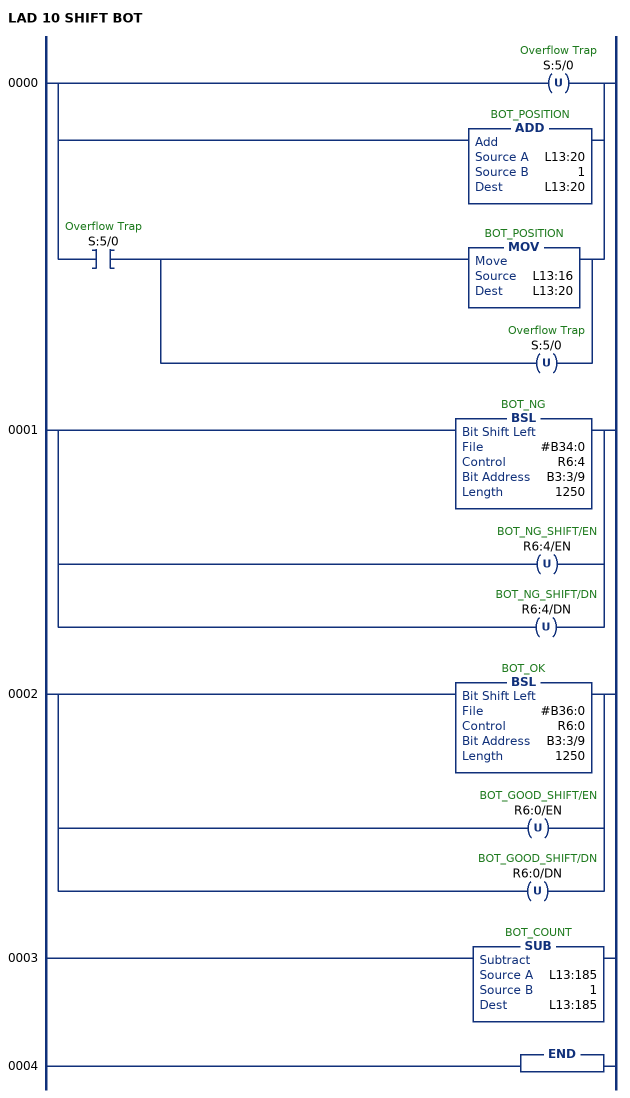
% Rung: 0 %
SOR BST OTU S:5/0 NXB ADD L13:20 1 L13:20 NXB XIC S:5/0 BST MOV L13:16 L13:20 NXB OTU S:5/0 BND BND EOR
%   S:5/0  "Overflow Trap" %
%   L13:20  BOT_POSITION %
%   L13:16  MIN_LONG %
% Rung: 1 %
SOR BST BSL #B34:0 R6:4 B3:3/9 1250 NXB OTU R6:4/EN NXB OTU R6:4/DN BND EOR
%   B34:0  BOT_NG %
%   R6:4  BOT_NG_SHIFT %
%   B3:3/9  OFF %
% Rung: 2 %
SOR BST BSL #B36:0 R6:0 B3:3/9 1250 NXB OTU R6:0/EN NXB OTU R6:0/DN BND EOR
%   B36:0  BOT_OK %
%   R6:0  BOT_GOOD_SHIFT %
%   B3:3/9  OFF %
% Rung: 3 %
SOR SUB L13:185 1 L13:185 EOR
%   L13:185  BOT_COUNT %
% Rung: 4 %
SOR END EOR

LADDER 11 "SHIFT TOP"
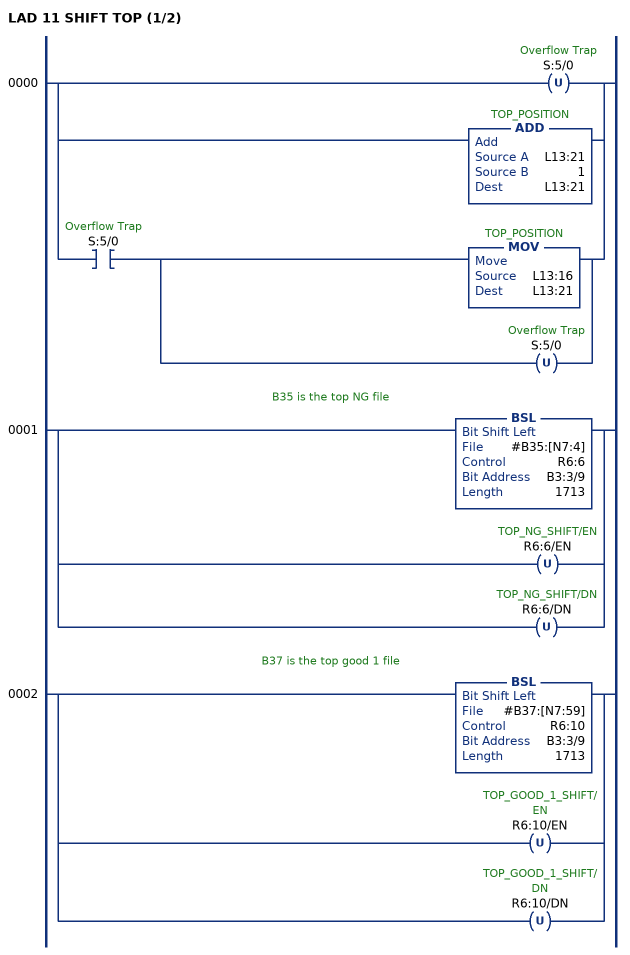
% Rung: 0 %
SOR BST OTU S:5/0 NXB ADD L13:21 1 L13:21 NXB XIC S:5/0 BST MOV L13:16 L13:21 NXB OTU S:5/0 BND BND EOR
%   S:5/0  "Overflow Trap" %
%   L13:21  TOP_POSITION %
%   L13:16  MIN_LONG %
% Rung: 1 %
% B35 is the top NG file %
SOR BST BSL #B35:[N7:4] R6:6 B3:3/9 1713 NXB OTU R6:6/EN NXB OTU R6:6/DN BND EOR
%   N7:4  TOP_NG_START_WORD %
%   R6:6  TOP_NG_SHIFT %
%   B3:3/9  OFF %
% Rung: 2 %
% B37 is the top good 1 file %
SOR BST BSL #B37:[N7:59] R6:10 B3:3/9 1713 NXB OTU R6:10/EN NXB OTU R6:10/DN BND EOR
%   N7:59  TOP_GOOD1_START_WORD %
%   R6:10  TOP_GOOD_1_SHIFT %
%   B3:3/9  OFF %

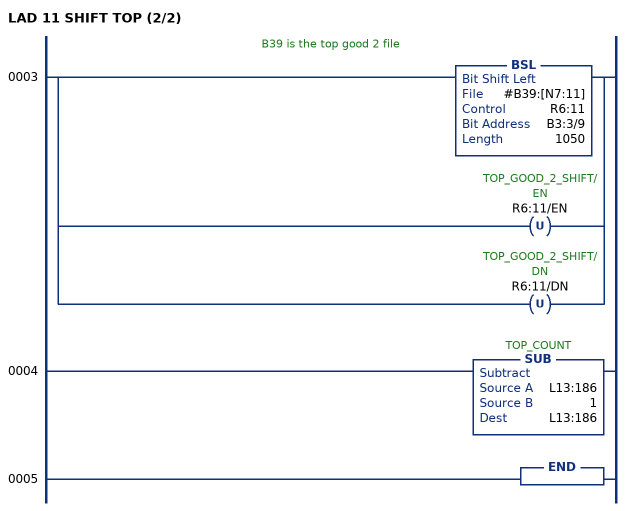
% Rung: 3 %
% B39 is the top good 2 file %
SOR BST BSL #B39:[N7:11] R6:11 B3:3/9 1050 NXB OTU R6:11/EN NXB OTU R6:11/DN BND EOR
%   N7:11  TOP_GOOD2_START_WORD %
%   R6:11  TOP_GOOD_2_SHIFT %
%   B3:3/9  OFF %
% Rung: 4 %
SOR SUB L13:186 1 L13:186 EOR
%   L13:186  TOP_COUNT %
% Rung: 5 %
SOR END EOR

LADDER 12 "BOTOPTIC"
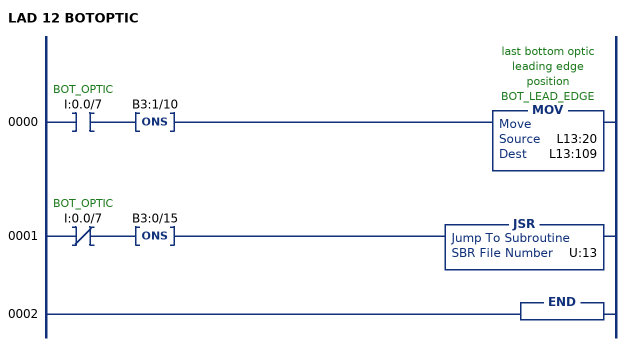
% Rung: 0 %
SOR XIC I:0.0/7 ONS B3:1/10 MOV L13:20 L13:109 EOR
%   I:0.0/7  BOT_OPTIC %
%   L13:20  BOT_POSITION %
%   L13:109  BOT_LEAD_EDGE  "last bottom optic leading edge position" %
% Rung: 1 %
SOR XIO I:0.0/7 ONS B3:0/15 JSR U:13 EOR
%   I:0.0/7  BOT_OPTIC %
% Rung: 2 %
SOR END EOR

LADDER 13 "BOTOPTMES"
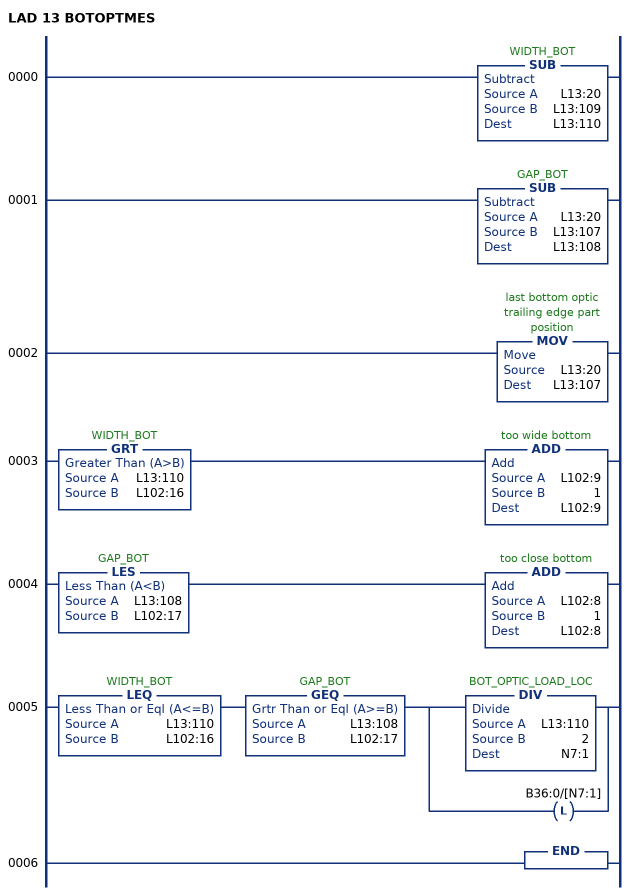
% Rung: 0 %
SOR SUB L13:20 L13:109 L13:110 EOR
%   L13:20  BOT_POSITION %
%   L13:109  BOT_LEAD_EDGE  "last bottom optic leading edge position" %
%   L13:110  WIDTH_BOT %
% Rung: 1 %
SOR SUB L13:20 L13:107 L13:108 EOR
%   L13:20  BOT_POSITION %
%   L13:107  "last bottom optic trailing edge part position" %
%   L13:108  GAP_BOT %
% Rung: 2 %
SOR MOV L13:20 L13:107 EOR
%   L13:20  BOT_POSITION %
%   L13:107  "last bottom optic trailing edge part position" %
% Rung: 3 %
SOR GRT L13:110 L102:16 ADD L102:9 1 L102:9 EOR
%   L13:110  WIDTH_BOT %
%   L102:16  BOT_MAX_WIDTH %
%   L102:9  "too wide bottom" %
% Rung: 4 %
SOR LES L13:108 L102:17 ADD L102:8 1 L102:8 EOR
%   L13:108  GAP_BOT %
%   L102:17  BOT_MIN_GAP %
%   L102:8  "too close bottom" %
% Rung: 5 %
SOR LEQ L13:110 L102:16 GEQ L13:108 L102:17 BST DIV L13:110 2 N7:1 NXB OTL B36:0/[N7:1] BND EOR
%   L13:110  WIDTH_BOT %
%   L102:16  BOT_MAX_WIDTH %
%   L13:108  GAP_BOT %
%   L102:17  BOT_MIN_GAP %
%   N7:1  BOT_OPTIC_LOAD_LOC %
%   B36:0  BOT_OK %
% Rung: 6 %
SOR END EOR

LADDER 14 "SHIFT TOP2"    % shift top inspection 6 %
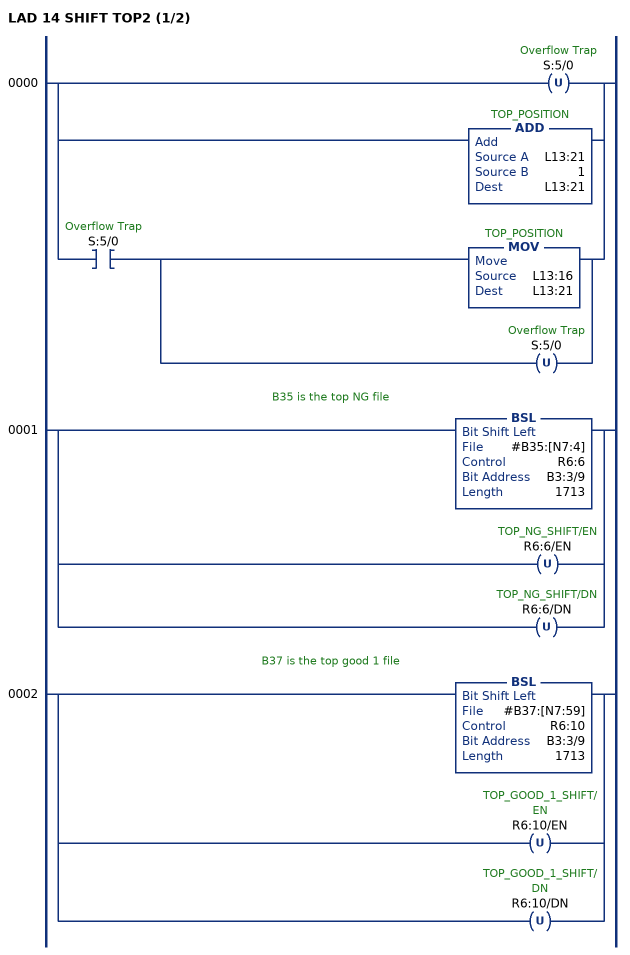
% Rung: 0 %
SOR BST OTU S:5/0 NXB ADD L13:21 1 L13:21 NXB XIC S:5/0 BST MOV L13:16 L13:21 NXB OTU S:5/0 BND BND EOR
%   S:5/0  "Overflow Trap" %
%   L13:21  TOP_POSITION %
%   L13:16  MIN_LONG %
% Rung: 1 %
% B35 is the top NG file %
SOR BST BSL #B35:[N7:4] R6:6 B3:3/9 1713 NXB OTU R6:6/EN NXB OTU R6:6/DN BND EOR
%   N7:4  TOP_NG_START_WORD %
%   R6:6  TOP_NG_SHIFT %
%   B3:3/9  OFF %
% Rung: 2 %
% B37 is the top good 1 file %
SOR BST BSL #B37:[N7:59] R6:10 B3:3/9 1713 NXB OTU R6:10/EN NXB OTU R6:10/DN BND EOR
%   N7:59  TOP_GOOD1_START_WORD %
%   R6:10  TOP_GOOD_1_SHIFT %
%   B3:3/9  OFF %

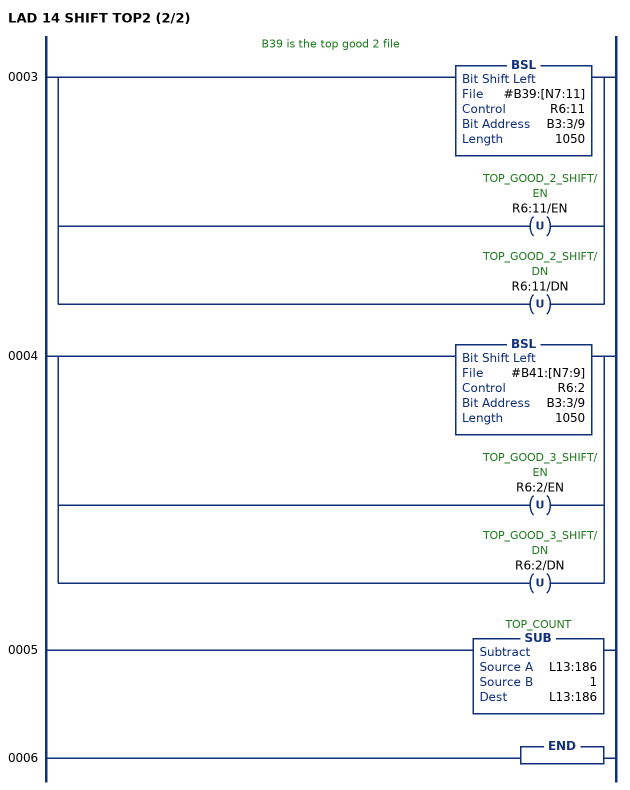
% Rung: 3 %
% B39 is the top good 2 file %
SOR BST BSL #B39:[N7:11] R6:11 B3:3/9 1050 NXB OTU R6:11/EN NXB OTU R6:11/DN BND EOR
%   N7:11  TOP_GOOD2_START_WORD %
%   R6:11  TOP_GOOD_2_SHIFT %
%   B3:3/9  OFF %
% Rung: 4 %
SOR BST BSL #B41:[N7:9] R6:2 B3:3/9 1050 NXB OTU R6:2/EN NXB OTU R6:2/DN BND EOR
%   N7:9  TOP_GOOD3_START_WORD %
%   R6:2  TOP_GOOD_3_SHIFT %
%   B3:3/9  OFF %
% Rung: 5 %
SOR SUB L13:186 1 L13:186 EOR
%   L13:186  TOP_COUNT %
% Rung: 6 %
SOR END EOR

LADDER 81 "I1"
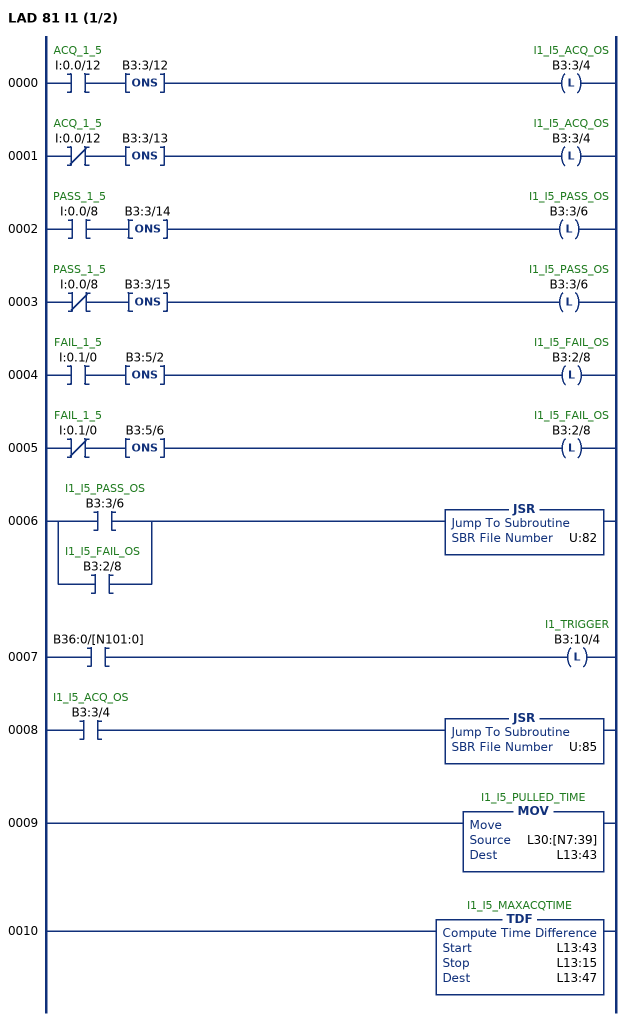
% Rung: 0 %
SOR XIC I:0.0/12 ONS B3:3/12 OTL B3:3/4 EOR
%   I:0.0/12  ACQ_1_5 %
%   B3:3/4  I1_I5_ACQ_OS %
% Rung: 1 %
SOR XIO I:0.0/12 ONS B3:3/13 OTL B3:3/4 EOR
%   I:0.0/12  ACQ_1_5 %
%   B3:3/4  I1_I5_ACQ_OS %
% Rung: 2 %
SOR XIC I:0.0/8 ONS B3:3/14 OTL B3:3/6 EOR
%   I:0.0/8  PASS_1_5 %
%   B3:3/6  I1_I5_PASS_OS %
% Rung: 3 %
SOR XIO I:0.0/8 ONS B3:3/15 OTL B3:3/6 EOR
%   I:0.0/8  PASS_1_5 %
%   B3:3/6  I1_I5_PASS_OS %
% Rung: 4 %
SOR XIC I:0.1/0 ONS B3:5/2 OTL B3:2/8 EOR
%   I:0.1/0  FAIL_1_5 %
%   B3:2/8  I1_I5_FAIL_OS %
% Rung: 5 %
SOR XIO I:0.1/0 ONS B3:5/6 OTL B3:2/8 EOR
%   I:0.1/0  FAIL_1_5 %
%   B3:2/8  I1_I5_FAIL_OS %
% Rung: 6 %
SOR BST XIC B3:3/6 NXB XIC B3:2/8 BND JSR U:82 EOR
%   B3:3/6  I1_I5_PASS_OS %
%   B3:2/8  I1_I5_FAIL_OS %
% Rung: 7 %
SOR XIC B36:0/[N101:0] OTL B3:10/4 EOR
%   B36:0  BOT_OK %
%   N101:0  I1_TRIG_LOC %
%   B3:10/4  I1_TRIGGER %
% Rung: 8 %
SOR XIC B3:3/4 JSR U:85 EOR
%   B3:3/4  I1_I5_ACQ_OS %
% Rung: 9 %
SOR MOV L30:[N7:39] L13:43 EOR
%   N7:39  I5_OLDEST_PART_INDEX %
%   L13:43  I1_I5_PULLED_TIME %
% Rung: 10 %
SOR TDF L13:43 L13:15 L13:47 EOR
%   L13:43  I1_I5_PULLED_TIME %
%   L13:15  THE_TIME %
%   L13:47  I1_I5_MAXACQTIME %

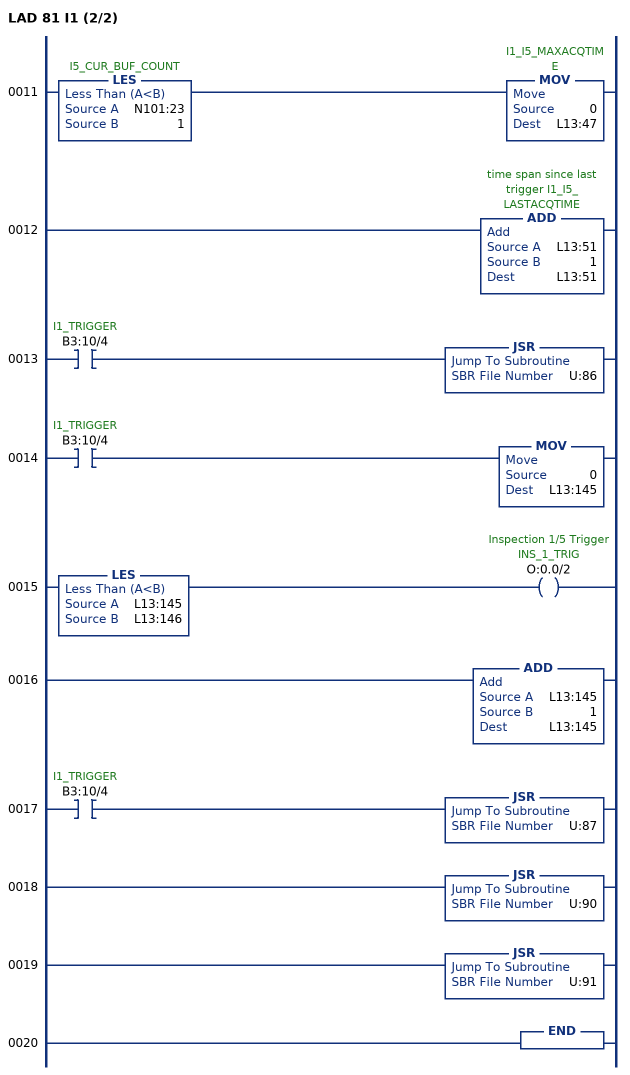
% Rung: 11 %
SOR LES N101:23 1 MOV 0 L13:47 EOR
%   N101:23  I5_CUR_BUF_COUNT %
%   L13:47  I1_I5_MAXACQTIME %
% Rung: 12 %
SOR ADD L13:51 1 L13:51 EOR
%   L13:51  I1_I5_LASTACQTIME  "time span since last trigger" %
% Rung: 13 %
SOR XIC B3:10/4 JSR U:86 EOR
%   B3:10/4  I1_TRIGGER %
% Rung: 14 %
SOR XIC B3:10/4 MOV 0 L13:145 EOR
%   B3:10/4  I1_TRIGGER %
% Rung: 15 %
SOR LES L13:145 L13:146 OTE O:0.0/2 EOR
%   O:0.0/2  INS_1_TRIG  "Inspection 1/5 Trigger" %
% Rung: 16 %
SOR ADD L13:145 1 L13:145 EOR
% Rung: 17 %
SOR XIC B3:10/4 JSR U:87 EOR
%   B3:10/4  I1_TRIGGER %
% Rung: 18 %
SOR JSR U:90 EOR
% Rung: 19 %
SOR JSR U:91 EOR
% Rung: 20 %
SOR END EOR

LADDER 82 "I1 RESULT"
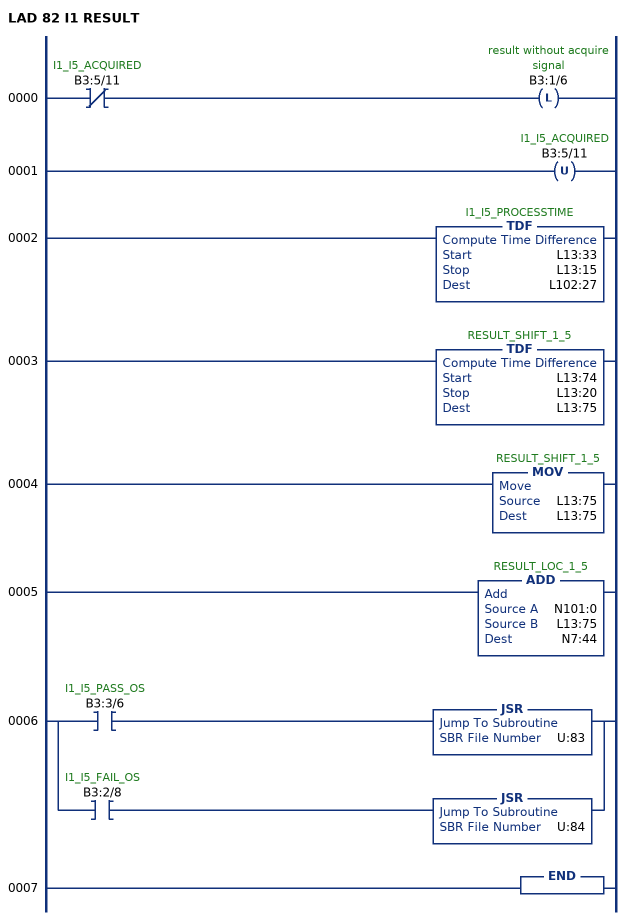
% Rung: 0 %
SOR XIO B3:5/11 OTL B3:1/6 EOR
%   B3:5/11  I1_I5_ACQUIRED %
%   B3:1/6  "result without acquire signal" %
% Rung: 1 %
SOR OTU B3:5/11 EOR
%   B3:5/11  I1_I5_ACQUIRED %
% Rung: 2 %
SOR TDF L13:33 L13:15 L102:27 EOR
%   L13:33  I1_I5_TIMEOFACQ %
%   L13:15  THE_TIME %
%   L102:27  I1_I5_PROCESSTIME %
% Rung: 3 %
SOR TDF L13:74 L13:20 L13:75 EOR
%   L13:74  I1_I5_PROC_START_POS %
%   L13:20  BOT_POSITION %
%   L13:75  RESULT_SHIFT_1_5 %
% Rung: 4 %
SOR MOV L13:75 L13:75 EOR
%   L13:75  RESULT_SHIFT_1_5 %
% Rung: 5 %
SOR ADD N101:0 L13:75 N7:44 EOR
%   N101:0  I1_TRIG_LOC %
%   L13:75  RESULT_SHIFT_1_5 %
%   N7:44  RESULT_LOC_1_5 %
% Rung: 6 %
SOR BST XIC B3:3/6 JSR U:83 NXB XIC B3:2/8 JSR U:84 BND EOR
%   B3:3/6  I1_I5_PASS_OS %
%   B3:2/8  I1_I5_FAIL_OS %
% Rung: 7 %
SOR END EOR

LADDER 83 "I1 PASS"
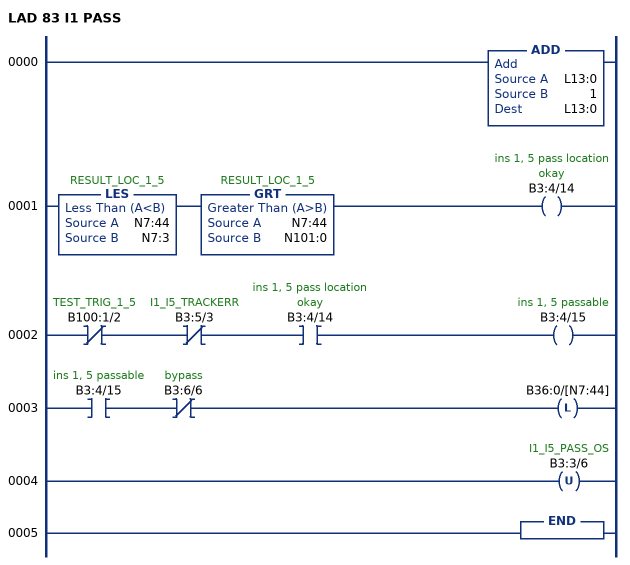
% Rung: 0 %
SOR ADD L13:0 1 L13:0 EOR
% Rung: 1 %
SOR LES N7:44 N7:3 GRT N7:44 N101:0 OTE B3:4/14 EOR
%   N7:44  RESULT_LOC_1_5 %
%   N7:3  I1_MAX_SHIFT %
%   N101:0  I1_TRIG_LOC %
%   B3:4/14  "ins 1, 5 pass location okay" %
% Rung: 2 %
SOR XIO B100:1/2 XIO B3:5/3 XIC B3:4/14 OTE B3:4/15 EOR
%   B100:1/2  TEST_TRIG_1_5 %
%   B3:5/3  I1_I5_TRACKERR %
%   B3:4/14  "ins 1, 5 pass location okay" %
%   B3:4/15  "ins 1, 5 passable" %
% Rung: 3 %
SOR XIC B3:4/15 XIO B3:6/6 OTL B36:0/[N7:44] EOR
%   B3:4/15  "ins 1, 5 passable" %
%   B3:6/6  "bypass" %
%   B36:0  BOT_OK %
%   N7:44  RESULT_LOC_1_5 %
% Rung: 4 %
SOR OTU B3:3/6 EOR
%   B3:3/6  I1_I5_PASS_OS %
% Rung: 5 %
SOR END EOR

LADDER 84 "I1 FAIL"
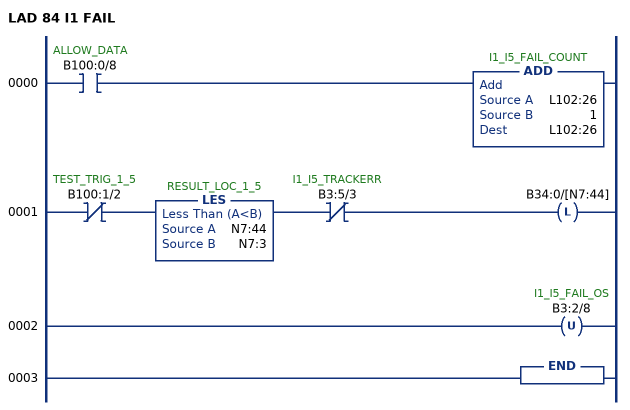
% Rung: 0 %
SOR XIC B100:0/8 ADD L102:26 1 L102:26 EOR
%   B100:0/8  ALLOW_DATA %
%   L102:26  I1_I5_FAIL_COUNT %
% Rung: 1 %
SOR XIO B100:1/2 LES N7:44 N7:3 XIO B3:5/3 OTL B34:0/[N7:44] EOR
%   B100:1/2  TEST_TRIG_1_5 %
%   N7:44  RESULT_LOC_1_5 %
%   N7:3  I1_MAX_SHIFT %
%   B3:5/3  I1_I5_TRACKERR %
%   B34:0  BOT_NG %
% Rung: 2 %
SOR OTU B3:2/8 EOR
%   B3:2/8  I1_I5_FAIL_OS %
% Rung: 3 %
SOR END EOR

LADDER 85 "I1 ACQ"
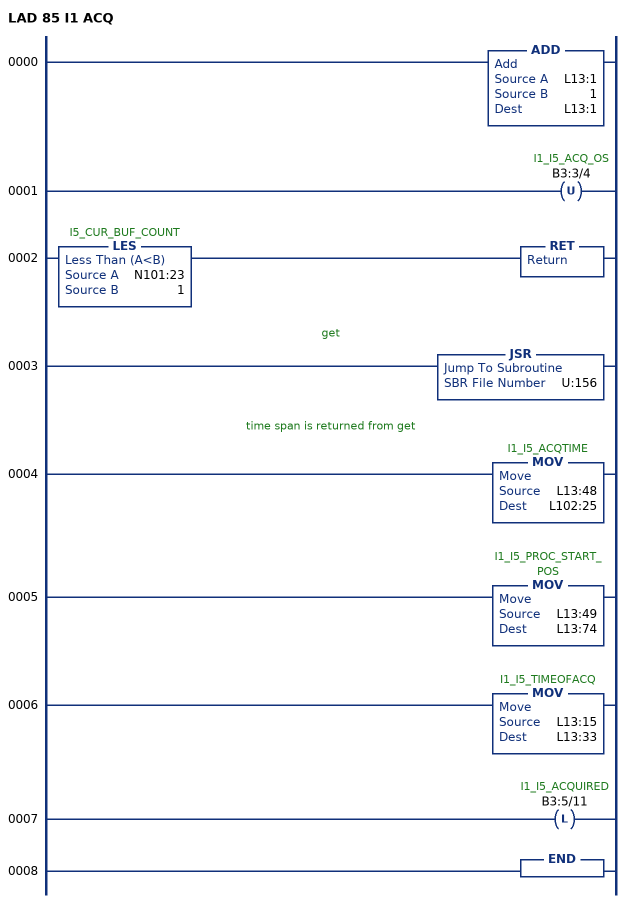
% Rung: 0 %
SOR ADD L13:1 1 L13:1 EOR
% Rung: 1 %
SOR OTU B3:3/4 EOR
%   B3:3/4  I1_I5_ACQ_OS %
% Rung: 2 %
SOR LES N101:23 1 RET EOR
%   N101:23  I5_CUR_BUF_COUNT %
% Rung: 3 %
% get %
SOR JSR U:156 EOR
% Rung: 4 %
% time span is returned from get %
SOR MOV L13:48 L102:25 EOR
%   L13:48  I1_I5_TIME_SPAN %
%   L102:25  I1_I5_ACQTIME %
% Rung: 5 %
SOR MOV L13:49 L13:74 EOR
%   L13:49  I1_I5_PULLED_POS %
%   L13:74  I1_I5_PROC_START_POS %
% Rung: 6 %
SOR MOV L13:15 L13:33 EOR
%   L13:15  THE_TIME %
%   L13:33  I1_I5_TIMEOFACQ %
% Rung: 7 %
SOR OTL B3:5/11 EOR
%   B3:5/11  I1_I5_ACQUIRED %
% Rung: 8 %
SOR END EOR

LADDER 86 "I1 TESTER"
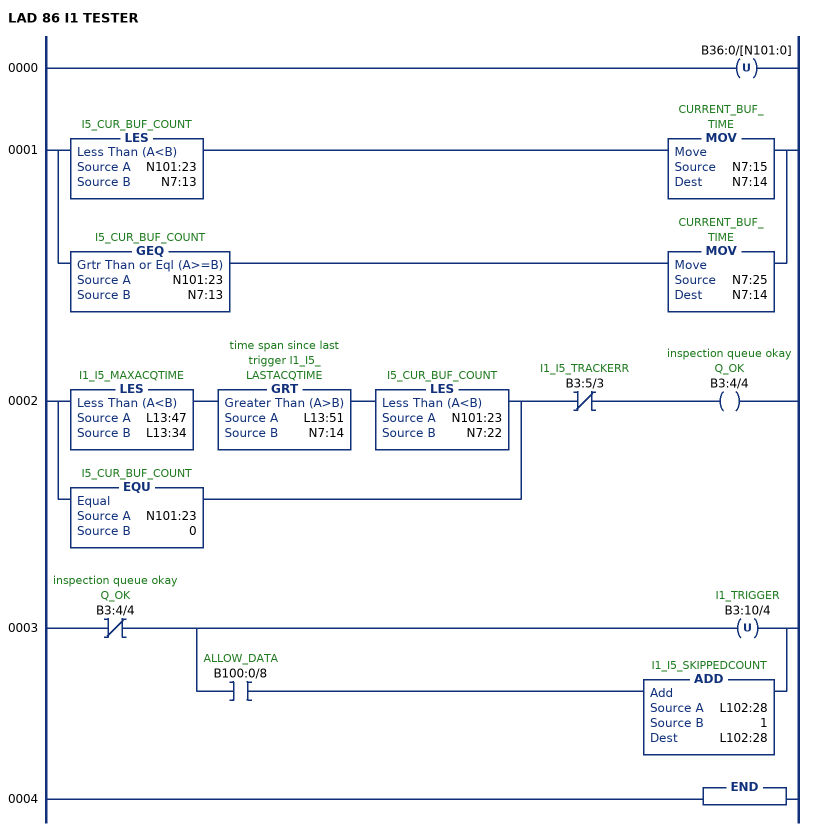
% Rung: 0 %
SOR OTU B36:0/[N101:0] EOR
%   B36:0  BOT_OK %
%   N101:0  I1_TRIG_LOC %
% Rung: 1 %
SOR BST LES N101:23 N7:13 MOV N7:15 N7:14 NXB GEQ N101:23 N7:13 MOV N7:25 N7:14 BND EOR
%   N101:23  I5_CUR_BUF_COUNT %
%   N7:13  BUF_TRANS  "cam to pc buf transition" %
%   N7:15  CAM_BUF_TIME  "cam buf time" %
%   N7:14  CURRENT_BUF_TIME %
%   N7:25  PC_BUF_TIME  "pc buf time" %
% Rung: 2 %
SOR BST LES L13:47 L13:34 GRT L13:51 N7:14 LES N101:23 N7:22 NXB EQU N101:23 0 BND XIO B3:5/3 OTE B3:4/4 EOR
%   L13:47  I1_I5_MAXACQTIME %
%   L13:34  MAX_ACQ_ALL  "absolute max acquire time before bypass trigger" %
%   L13:51  I1_I5_LASTACQTIME  "time span since last trigger" %
%   N7:14  CURRENT_BUF_TIME %
%   N101:23  I5_CUR_BUF_COUNT %
%   N7:22  MAX_BUF_ALL  "max buffer count alowed before bypass" %
%   B3:5/3  I1_I5_TRACKERR %
%   B3:4/4  Q_OK  "inspection queue okay" %
% Rung: 3 %
SOR XIO B3:4/4 BST OTU B3:10/4 NXB XIC B100:0/8 ADD L102:28 1 L102:28 BND EOR
%   B3:4/4  Q_OK  "inspection queue okay" %
%   B3:10/4  I1_TRIGGER %
%   B100:0/8  ALLOW_DATA %
%   L102:28  I1_I5_SKIPPEDCOUNT %
% Rung: 4 %
SOR END EOR

LADDER 87 "I1 TRIG"
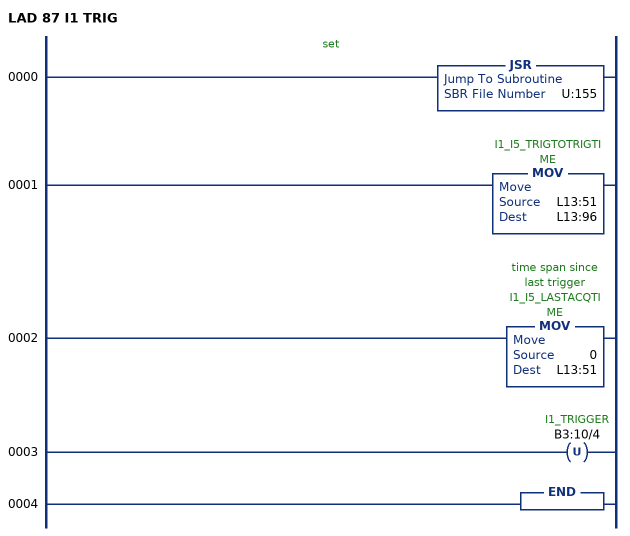
% Rung: 0 %
% set %
SOR JSR U:155 EOR
% Rung: 1 %
SOR MOV L13:51 L13:96 EOR
%   L13:51  I1_I5_LASTACQTIME  "time span since last trigger" %
%   L13:96  I1_I5_TRIGTOTRIGTIME %
% Rung: 2 %
SOR MOV 0 L13:51 EOR
%   L13:51  I1_I5_LASTACQTIME  "time span since last trigger" %
% Rung: 3 %
SOR OTU B3:10/4 EOR
%   B3:10/4  I1_TRIGGER %
% Rung: 4 %
SOR END EOR

LADDER 90 "I1 DATA"
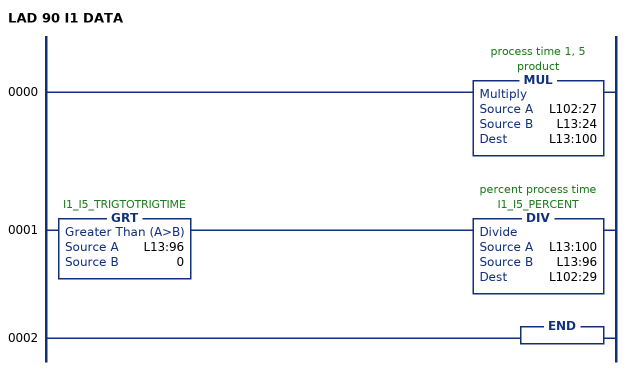
% Rung: 0 %
SOR MUL L102:27 L13:24 L13:100 EOR
%   L102:27  I1_I5_PROCESSTIME %
%   L13:24  "multiplyer to make devision come out to a percentage" %
%   L13:100  "process time 1, 5 product" %
% Rung: 1 %
SOR GRT L13:96 0 DIV L13:100 L13:96 L102:29 EOR
%   L13:96  I1_I5_TRIGTOTRIGTIME %
%   L13:100  "process time 1, 5 product" %
%   L102:29  I1_I5_PERCENT  "percent process time" %
% Rung: 2 %
SOR END EOR

LADDER 91 "I1 FAULT"
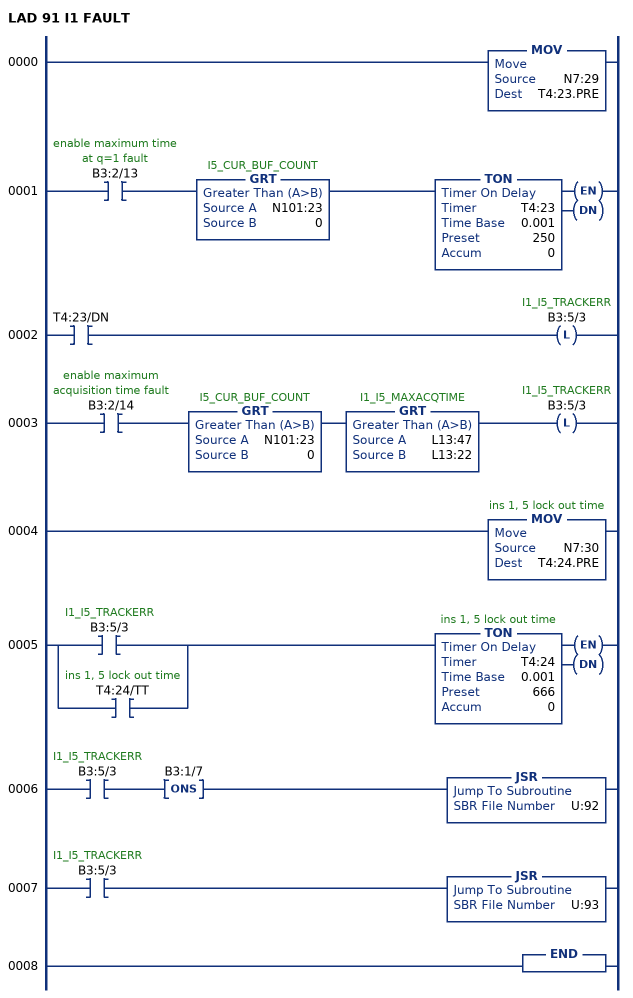
% Rung: 0 %
SOR MOV N7:29 T4:23.PRE EOR
%   N7:29  "max allowed ms time for q to be above 1 if safe fault is used" %
% Rung: 1 %
SOR XIC B3:2/13 GRT N101:23 0 TON T4:23 0.001 250 0 EOR
%   B3:2/13  "enable maximum time at q=1 fault" %
%   N101:23  I5_CUR_BUF_COUNT %
% Rung: 2 %
SOR XIC T4:23/DN OTL B3:5/3 EOR
%   B3:5/3  I1_I5_TRACKERR %
% Rung: 3 %
SOR XIC B3:2/14 GRT N101:23 0 GRT L13:47 L13:22 OTL B3:5/3 EOR
%   B3:2/14  "enable maximum acquisition time fault" %
%   N101:23  I5_CUR_BUF_COUNT %
%   L13:47  I1_I5_MAXACQTIME %
%   L13:22  "maximum of the longest acquire time allowed if maximum acquire time fault is enabled" %
%   B3:5/3  I1_I5_TRACKERR %
% Rung: 4 %
SOR MOV N7:30 T4:24.PRE EOR
%   N7:30  "ms time setting to lock out inspection to give all pending images a chance to clear" %
%   T4:24  "ins 1, 5 lock out time" %
% Rung: 5 %
SOR BST XIC B3:5/3 NXB XIC T4:24/TT BND TON T4:24 0.001 666 0 EOR
%   B3:5/3  I1_I5_TRACKERR %
%   T4:24  "ins 1, 5 lock out time" %
% Rung: 6 %
SOR XIC B3:5/3 ONS B3:1/7 JSR U:92 EOR
%   B3:5/3  I1_I5_TRACKERR %
% Rung: 7 %
SOR XIC B3:5/3 JSR U:93 EOR
%   B3:5/3  I1_I5_TRACKERR %
% Rung: 8 %
SOR END EOR

LADDER 92 "I1 FIX1"
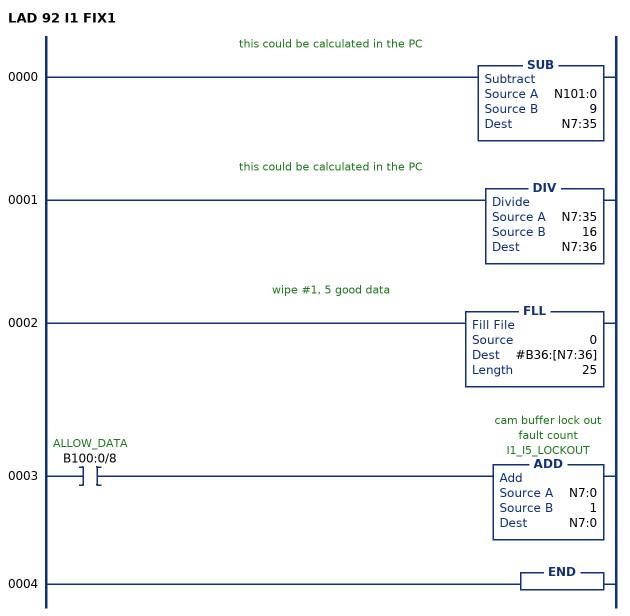
% Rung: 0 %
% this could be calculated in the PC %
SOR SUB N101:0 9 N7:35 EOR
%   N101:0  I1_TRIG_LOC %
% Rung: 1 %
% this could be calculated in the PC %
SOR DIV N7:35 16 N7:36 EOR
% Rung: 2 %
% wipe #1, 5 good data %
SOR FLL 0 #B36:[N7:36] 25 EOR
% Rung: 3 %
SOR XIC B100:0/8 ADD N7:0 1 N7:0 EOR
%   B100:0/8  ALLOW_DATA %
%   N7:0  I1_I5_LOCKOUT  "cam buffer lock out fault count" %
% Rung: 4 %
SOR END EOR

LADDER 93 "I1 FIX2"
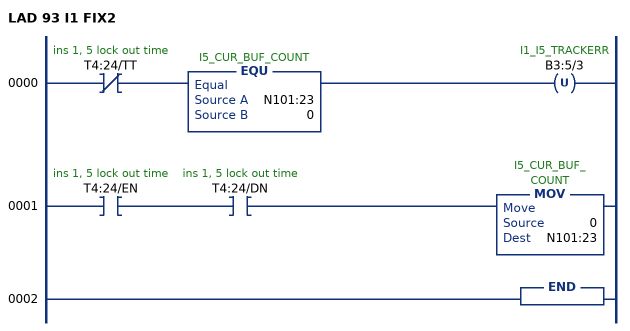
% Rung: 0 %
SOR XIO T4:24/TT EQU N101:23 0 OTU B3:5/3 EOR
%   T4:24  "ins 1, 5 lock out time" %
%   N101:23  I5_CUR_BUF_COUNT %
%   B3:5/3  I1_I5_TRACKERR %
% Rung: 1 %
SOR XIC T4:24/EN XIC T4:24/DN MOV 0 N101:23 EOR
%   T4:24  "ins 1, 5 lock out time" %
%   N101:23  I5_CUR_BUF_COUNT %
% Rung: 2 %
SOR END EOR

LADDER 135 "XFER"
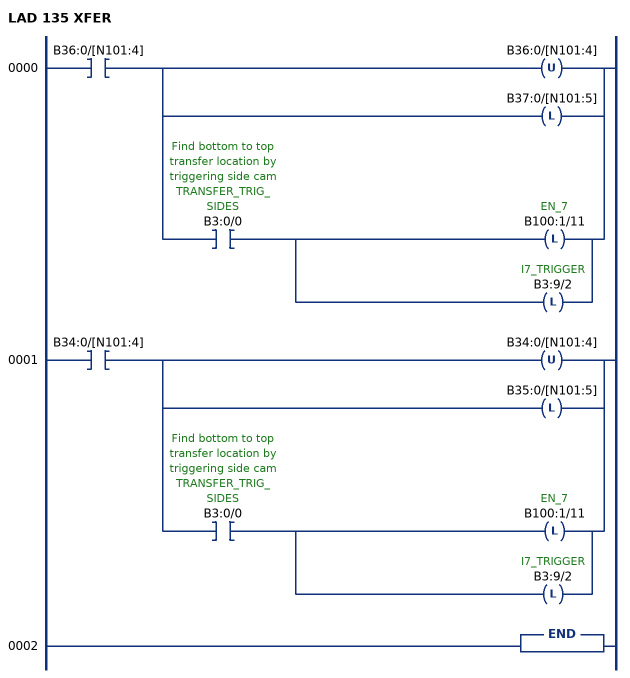
% Rung: 0 %
SOR XIC B36:0/[N101:4] BST OTU B36:0/[N101:4] NXB OTL B37:0/[N101:5] NXB XIC B3:0/0 BST OTL B100:1/11 NXB OTL B3:9/2 BND BND EOR
%   B36:0  BOT_OK %
%   N101:4  XFER_OUT_LOC %
%   B37:0  TOP_OK_1 %
%   N101:5  XFER_IN_LOC %
%   B3:0/0  TRANSFER_TRIG_SIDES  "Find bottom to top transfer location by triggering side cam" %
%   B100:1/11  EN_7 %
%   B3:9/2  I7_TRIGGER %
% Rung: 1 %
SOR XIC B34:0/[N101:4] BST OTU B34:0/[N101:4] NXB OTL B35:0/[N101:5] NXB XIC B3:0/0 BST OTL B100:1/11 NXB OTL B3:9/2 BND BND EOR
%   B34:0  BOT_NG %
%   N101:4  XFER_OUT_LOC %
%   B35:0  TOP_NG %
%   N101:5  XFER_IN_LOC %
%   B3:0/0  TRANSFER_TRIG_SIDES  "Find bottom to top transfer location by triggering side cam" %
%   B100:1/11  EN_7 %
%   B3:9/2  I7_TRIGGER %
% Rung: 2 %
SOR END EOR

LADDER 137 "TOPOPTIC"
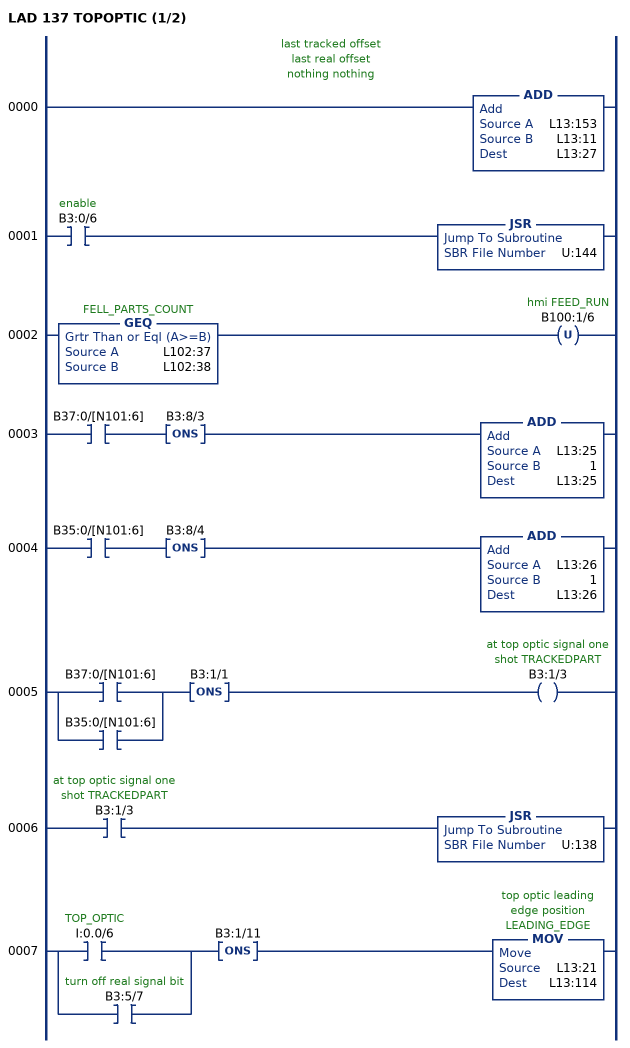
% Rung: 0 %
% last tracked offset
% last real offset
% nothing nothing %
SOR ADD L13:153 L13:11 L13:27 EOR
%   L13:153  NORM_VERT_OFFSET  "normal alignment offset at vertual abs L13:152" %
%   L13:11  NORM_REAL_OFFSET  "normal alignment offset at real abs L13:154" %
% Rung: 1 %
SOR XIC B3:0/6 JSR U:144 EOR
%   B3:0/6  "enable" %
% Rung: 2 %
SOR GEQ L102:37 L102:38 OTU B100:1/6 EOR
%   L102:37  FELL_PARTS_COUNT %
%   L102:38  FELL_PARTS_LIMIT %
%   B100:1/6  FEED_RUN  "hmi" %
% Rung: 3 %
SOR XIC B37:0/[N101:6] ONS B3:8/3 ADD L13:25 1 L13:25 EOR
%   B37:0  TOP_OK_1 %
%   N101:6  TOP_OPTIC_LOC %
% Rung: 4 %
SOR XIC B35:0/[N101:6] ONS B3:8/4 ADD L13:26 1 L13:26 EOR
%   B35:0  TOP_NG %
%   N101:6  TOP_OPTIC_LOC %
% Rung: 5 %
SOR BST XIC B37:0/[N101:6] NXB XIC B35:0/[N101:6] BND ONS B3:1/1 OTE B3:1/3 EOR
%   B37:0  TOP_OK_1 %
%   N101:6  TOP_OPTIC_LOC %
%   B35:0  TOP_NG %
%   B3:1/3  TRACKEDPART  "at top optic signal one shot" %
% Rung: 6 %
SOR XIC B3:1/3 JSR U:138 EOR
%   B3:1/3  TRACKEDPART  "at top optic signal one shot" %
% Rung: 7 %
SOR BST XIC I:0.0/6 NXB XIC B3:5/7 BND ONS B3:1/11 MOV L13:21 L13:114 EOR
%   I:0.0/6  TOP_OPTIC %
%   B3:5/7  "turn off real signal bit" %
%   L13:21  TOP_POSITION %
%   L13:114  LEADING_EDGE  "top optic leading edge position" %

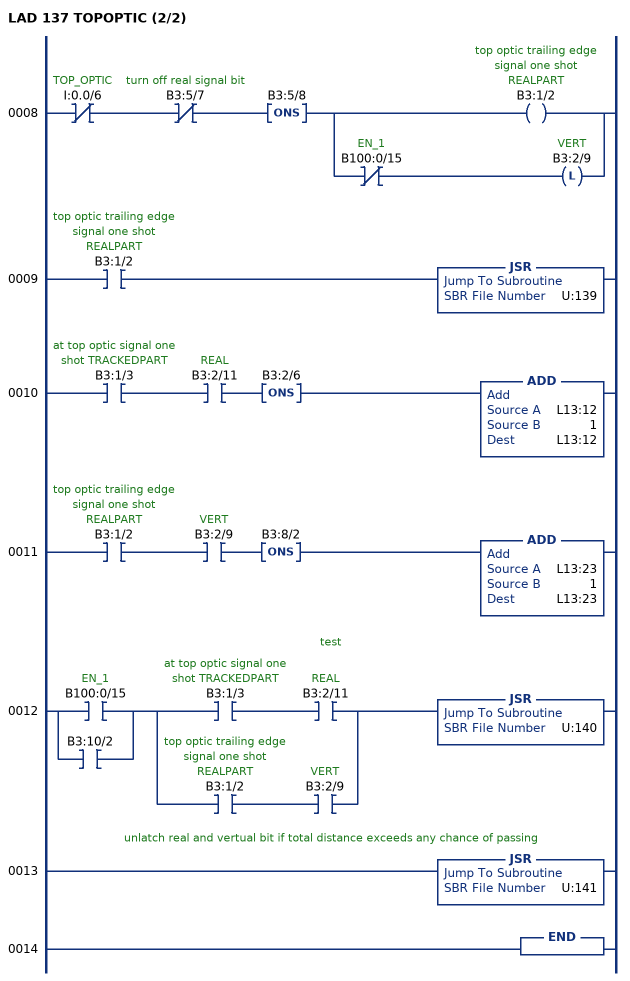
% Rung: 8 %
SOR XIO I:0.0/6 XIO B3:5/7 ONS B3:5/8 BST OTE B3:1/2 NXB XIO B100:0/15 OTL B3:2/9 BND EOR
%   I:0.0/6  TOP_OPTIC %
%   B3:5/7  "turn off real signal bit" %
%   B3:1/2  REALPART  "top optic trailing edge signal one shot" %
%   B100:0/15  EN_1 %
%   B3:2/9  VERT %
% Rung: 9 %
SOR XIC B3:1/2 JSR U:139 EOR
%   B3:1/2  REALPART  "top optic trailing edge signal one shot" %
% Rung: 10 %
SOR XIC B3:1/3 XIC B3:2/11 ONS B3:2/6 ADD L13:12 1 L13:12 EOR
%   B3:1/3  TRACKEDPART  "at top optic signal one shot" %
%   B3:2/11  REAL %
% Rung: 11 %
SOR XIC B3:1/2 XIC B3:2/9 ONS B3:8/2 ADD L13:23 1 L13:23 EOR
%   B3:1/2  REALPART  "top optic trailing edge signal one shot" %
%   B3:2/9  VERT %
% Rung: 12 %
% test %
SOR BST XIC B100:0/15 NXB XIC B3:10/2 BND BST XIC B3:1/3 XIC B3:2/11 NXB XIC B3:1/2 XIC B3:2/9 BND JSR U:140 EOR
%   B100:0/15  EN_1 %
%   B3:1/3  TRACKEDPART  "at top optic signal one shot" %
%   B3:2/11  REAL %
%   B3:1/2  REALPART  "top optic trailing edge signal one shot" %
%   B3:2/9  VERT %
% Rung: 13 %
% unlatch real and vertual bit if total distance exceeds any chance of passing %
SOR JSR U:141 EOR
% Rung: 14 %
SOR END EOR

LADDER 138 "TOPOPVERT"
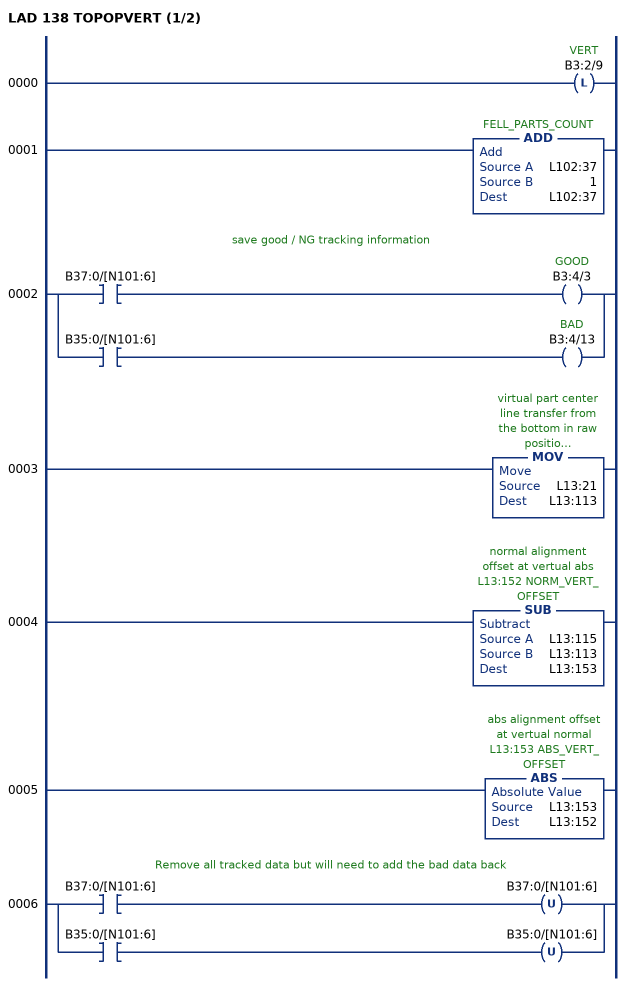
% Rung: 0 %
SOR OTL B3:2/9 EOR
%   B3:2/9  VERT %
% Rung: 1 %
SOR ADD L102:37 1 L102:37 EOR
%   L102:37  FELL_PARTS_COUNT %
% Rung: 2 %
% save good / NG tracking information %
SOR BST XIC B37:0/[N101:6] OTE B3:4/3 NXB XIC B35:0/[N101:6] OTE B3:4/13 BND EOR
%   B37:0  TOP_OK_1 %
%   N101:6  TOP_OPTIC_LOC %
%   B3:4/3  GOOD %
%   B35:0  TOP_NG %
%   B3:4/13  BAD %
% Rung: 3 %
SOR MOV L13:21 L13:113 EOR
%   L13:21  TOP_POSITION %
%   L13:113  VERTUAL_PT_RAW_CL  "virtual part center line transfer from the bottom in raw position" %
% Rung: 4 %
SOR SUB L13:115 L13:113 L13:153 EOR
%   L13:115  TRAILING_EDGE_RAW  "top optic trailing edge position" %
%   L13:113  VERTUAL_PT_RAW_CL  "virtual part center line transfer from the bottom in raw position" %
%   L13:153  NORM_VERT_OFFSET  "normal alignment offset at vertual abs L13:152" %
% Rung: 5 %
SOR ABS L13:153 L13:152 EOR
%   L13:153  NORM_VERT_OFFSET  "normal alignment offset at vertual abs L13:152" %
%   L13:152  ABS_VERT_OFFSET  "abs alignment offset at vertual normal L13:153" %
% Rung: 6 %
% Remove all tracked data but will need to add the bad data back %
SOR BST XIC B37:0/[N101:6] OTU B37:0/[N101:6] NXB XIC B35:0/[N101:6] OTU B35:0/[N101:6] BND EOR
%   B37:0  TOP_OK_1 %
%   N101:6  TOP_OPTIC_LOC %
%   B35:0  TOP_NG %

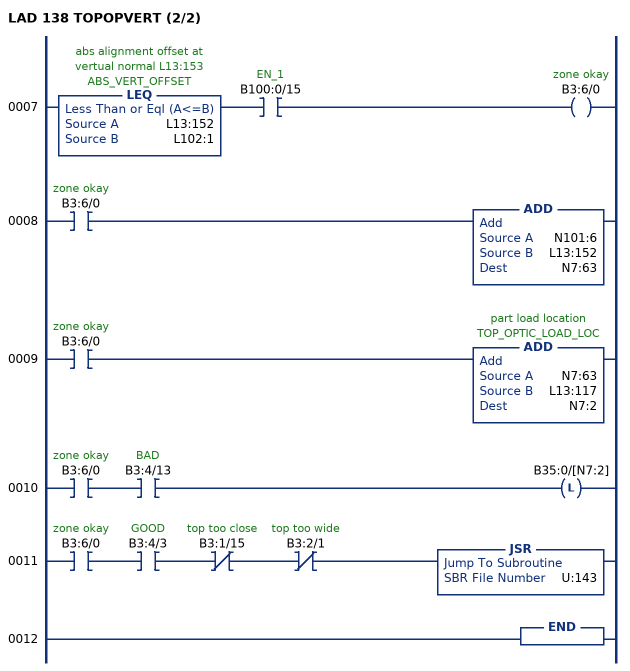
% Rung: 7 %
SOR LEQ L13:152 L102:1 XIC B100:0/15 OTE B3:6/0 EOR
%   L13:152  ABS_VERT_OFFSET  "abs alignment offset at vertual normal L13:153" %
%   L102:1  MAX_OFFSET  "transition zone width" %
%   B100:0/15  EN_1 %
%   B3:6/0  "zone okay" %
% Rung: 8 %
SOR XIC B3:6/0 ADD N101:6 L13:152 N7:63 EOR
%   B3:6/0  "zone okay" %
%   N101:6  TOP_OPTIC_LOC %
%   L13:152  ABS_VERT_OFFSET  "abs alignment offset at vertual normal L13:153" %
% Rung: 9 %
SOR XIC B3:6/0 ADD N7:63 L13:117 N7:2 EOR
%   B3:6/0  "zone okay" %
%   L13:117  HALF_WIDTH  "1/2 width top" %
%   N7:2  TOP_OPTIC_LOAD_LOC  "part load location" %
% Rung: 10 %
SOR XIC B3:6/0 XIC B3:4/13 OTL B35:0/[N7:2] EOR
%   B3:6/0  "zone okay" %
%   B3:4/13  BAD %
%   B35:0  TOP_NG %
%   N7:2  TOP_OPTIC_LOAD_LOC  "part load location" %
% Rung: 11 %
SOR XIC B3:6/0 XIC B3:4/3 XIO B3:1/15 XIO B3:2/1 JSR U:143 EOR
%   B3:6/0  "zone okay" %
%   B3:4/3  GOOD %
%   B3:1/15  "top too close" %
%   B3:2/1  "top too wide" %
% Rung: 12 %
SOR END EOR

LADDER 139 "TOPOPREAL"
